// TwinCAT 3 PLC project DomeRunTime
// ProgramVersion: 3.1.4023.0
// libraries:
//   Tc2_Standard, * (Beckhoff Automation GmbH)
//   Tc2_System, * (Beckhoff Automation GmbH)
//   Tc2_Utilities, * (Beckhoff Automation GmbH)
//   Tc3_Module, * (Beckhoff Automation GmbH)
//   Tc2_SystemCX,3.3.6.0,Beckhoff Automation GmbH
// project tree:
//   GVLs/ GVL_Dome.TcGVL
//   / PlcTask.TcTTO
//   POUs/ FB_EventLog.TcPOU, MAIN.TcPOU, NewADSRoute.TcPOU
// real-time tasks:
//   TASK PlcTask: cycle T#10ms, priority 20, ADS port 350
// I/O:
//   DEVICE Gerät 2 (EtherCAT), AmsNetId 5.73.45.158.3.1
//     Klemme 1 (EK1200) [EK1200-5000 EtherCAT Netzteil (2A E-Bus)]
//       Klemme 2 (EL6021) [EL6021 Schnittstelle (RS422/485)]
//       Klemme 3 (EL2008) [EL2008 8K. Dig. Ausgang 24V, 0.5A]
//       Klemme 4 (EL1008) [EL1008 8K. Dig. Eingang 24V, 3ms]
//       Klemme 5 (EL9011) [EL9011 Endklemme]
// variable links:
//   DomeRunTime/DomeRunTime Instance <-> Device 2 (EtherCAT)/Term 1 (EK1200)/Term 3 (EL2008)
//     PlcTask Outputs/GVL_Dome.Flap_enable <-> Channel 1/Output
//     PlcTask Outputs/GVL_Dome.Flap_open <-> Channel 2/Output
//     PlcTask Outputs/GVL_Dome.Slit_enable <-> Channel 3/Output
//     PlcTask Outputs/GVL_Dome.slit_open <-> Channel 4/Output
//   DomeRunTime/DomeRunTime Instance <-> Device 2 (EtherCAT)/Term 1 (EK1200)/Term 4 (EL1008)
//     PlcTask Inputs/GVL_Dome.Input7 <-> Channel 7/Input

CONFIGURATION DomeRunTime
    RESOURCE PLC ON TwinCAT3
        TASK PlcTask(INTERVAL := T#10ms, PRIORITY := 20);
        PROGRAM MAIN WITH PlcTask : MAIN;
    END_RESOURCE
END_CONFIGURATION

// ---- GVLs/GVL_Dome.TcGVL
{attribute 'qualified_only'}
VAR_GLOBAL
	// enable flap hydraulics
	Flap_enable		AT%Q*:	BOOL;
	// open the flap, when true; close when false
	Flap_open		AT%Q*:	BOOL;
	// enable the slit motor
	Slit_enable		AT%Q*:	BOOL;
	// open the slit when true; close when false
	slit_open		AT%Q*:	BOOL;
	// Input signal 7 (0...7)
	Input7		AT%I*: BOOL;

	// ADS remote control word
	StatusWord		AT%MW0: WORD;
END_VAR

// ---- POUs/MAIN.TcPOU
PROGRAM MAIN
VAR
	// open flap command
	OpenFlap:	BOOL;
	// close flap command
	CloseFlap:	BOOL;
	// open slit command
	OpenSlit:	BOOL;
	// close slit command
	CloseSlit:	BOOL;
	// flap open state
	FlapOpen:	BOOL := TRUE; // assume Flap Open after restart
	// flap closed state
	FlapClosed:	BOOL := FALSE;
	// slit open state
	SlitOpen:	BOOL := TRUE; // assume Slit Open after restart
	// slit closed state
	SlitClosed:	BOOL := FALSE;
	// assume dome open, after power loss / reboot
	DomeOpen:	BOOL := FALSE;
	// dome closed state
	DomeClosed:	BOOL := FALSE;
	// control word is valid
	Valid:		BOOL;
	// timer to delay the flap
	FlapDelay: TON;
	// timer to delay the slit on reverse of direction
	SlitDelay:	TON;
	FlapTimer,
	SlitTimer:	TP := (PT := T#60S);
	FlapDone,
	SlitDone:	F_TRIG;
	SyncOut:	TON;
	TimeOut:	TON;
	WD_LED:		E_CX81x0_LED;
	ERR_LED:	E_CX81x0_LED;
	DomeOpenEvent:		FB_EventLog;
	DomeClosedEvent:	FB_EventLog;
	SyncEvent:		FB_Eventlog;
	TimeoutEvent:	FB_Eventlog;
	ADSErrorEvent:	FB_Eventlog;
	ReadCycle:	TON := (PT:=T#100MS);
	fbReadReq:	ADSREAD := ( NETID := '5.78.96.50.1.1', PORT := 851, TMOUT := DEFAULT_ADS_TIMEOUT );
	ControlWord: 	WORD;
	Busy:	BOOL;
	ADSError:	BOOL;
	ADSErrorID: UDINT;
END_VAR

(*
Dome Control Remote Unit CX8190
########################

The dome is controlled by the main PLC using the GVL_Dome.ControlWord,
which is used to exchange commands to open and close the slit and the flap
and to report wether the dome is open or closed.
*)
//NewADSRoute();
ReadCycle(IN := TRUE);
IF ReadCycle.Q THEN
	// read if the ADS command is busy
	fbReadReq(	READ := FALSE,
				BUSY => Busy,
				ERR =>	ADSError,
				ERRID => ADSErrorID);
	IF NOT Busy THEN
		fbReadReq(  IDXGRP := 16#4020, 
					IDXOFFS := 0, 
					LEN := SIZEOF(ControlWord), 
					DESTADDR := ADR(ControlWord),
					READ := TRUE,
					BUSY => Busy,
					ERR =>	ADSError,
					ERRID => ADSErrorID);
		ReadCycle(IN := FALSE);
	ELSE
		// reset the read command
		fbReadReq(READ := FALSE);
	END_IF
	IF NOT ADSError THEN // we have valid data
		Valid := 	ControlWord.0;
		OpenFlap := ControlWord.1;
		OpenSlit := ControlWord.2;
		CloseFlap := NOT ControlWord.1;
		CloseSlit := NOT ControlWord.2;
		ERR_LED := E_CX81x0_LED.eCX81x0_LED_RED_OFF;
	ELSE
		// reset the control word
		ControlWord := 0;
	END_IF
	
END_IF

// This is the sync timeout. If we loose the sync for 5 seconds, we issue a warning.
SyncOut(IN := NOT Valid, PT := T#5S);
IF SyncOut.Q THEN
	ERR_LED := E_CX81x0_LED.eCX81x0_LED_RED_FLASHING_200ms;
END_IF

// This is the watchdog timer. If we don't get a valid signal within n seconds, we issue to close the dome.
TimeOut(IN := NOT Valid, PT := T#30S);
IF TimeOut.Q THEN
	CloseFlap := NOT FlapClosed;
	CloseSlit := NOT SlitClosed;
	ERR_LED := E_CX81x0_LED.eCX81x0_LED_RED_ON;
END_IF

// cancel commands, if we know that the slot is closed
IF SlitClosed AND CloseSlit THEN
	CloseSlit := FALSE;
END_IF
IF SlitOpen AND OpenSlit THEN
	OpenSlit := FALSE;
END_IF
IF FlapClosed AND CloseFlap THEN
	CloseFlap := FALSE;
END_IF
IF FlapOpen AND OpenFlap THEN
	OpenFlap := FALSE;
END_IF

IF CloseSlit AND SlitTimer.Q THEN
	OpenSlit := FALSE;
	GVL_Dome.Slit_open := FALSE;
	WD_LED := E_CX81x0_LED.eCX81x0_LED_GREEN_FLASHING_500ms;
END_IF

IF OpenSlit AND SlitTimer.Q THEN
	GVL_Dome.Slit_open := TRUE;
	WD_LED := E_CX81x0_LED.eCX81x0_LED_RED_FLASHING_500ms;
END_IF

IF CloseFlap AND FlapTimer.Q  THEN
	OpenFlap := FALSE;
	GVL_Dome.Flap_open := FALSE;
	WD_LED := E_CX81x0_LED.eCX81x0_LED_GREEN_FLASHING_200ms;
END_IF

IF OpenFlap AND FlapTimer.Q THEN
	GVL_Dome.Flap_open := TRUE;
	WD_LED := E_CX81x0_LED.eCX81x0_LED_RED_FLASHING_200ms;
END_IF

// if we reverse the direction of the flap, wait n milliseconds, otherwise we blow the fuse
FlapDelay(  IN := OpenFlap OR CloseFlap,
			PT := T#1000MS);
// After an initial delay, enable the signal for n seconds to move the flap.
// we have to use different times for opening and closing especially at low temperatures
IF OpenFlap THEN
	FlapTimer.PT := T#30S;
ELSIF CloseFlap THEN
	FlapTimer.PT := T#60S;
END_IF			
FlapTimer(  IN := FlapDelay.Q,
			Q => GVL_Dome.Flap_enable);
// a falling edge of the enable signal indicates, that we are done
FlapDone(CLK := GVL_Dome.Flap_enable);
// deactivate open or close signal if enable becomes false;
IF FlapDone.Q THEN
	IF OpenFlap THEN
		FlapOpen 	:= TRUE;
		FlapClosed 	:= FALSE;
	ELSIF CloseFlap THEN
		FlapClosed 	:= TRUE;
		FlapOpen 	:= FALSE;
	END_IF
	OpenFlap := FALSE;
	CloseFlap := FALSE;
END_IF
			
// if we reverse the direction of the flap, wait n milliseconds, otherwise we blow the fuse
SlitDelay(  IN := OpenSlit OR CloseSlit, 
			PT := T#1000MS); 

// After an initial delay, enable the signal for n seconds to move the slit.			
SlitTimer(  IN := SlitDelay.Q,
			PT := T#70S,
			Q => GVL_Dome.Slit_enable); 
// a falling edge of the enable signal indicates, that we are done			
SlitDone(CLK := GVL_Dome.Slit_enable);

IF SlitDone.Q THEN
	IF OpenSlit THEN
		SlitOpen := TRUE;
		SlitClosed := FALSE;
	ELSIF CloseSlit THEN
		SlitClosed := TRUE;
		SlitOpen := FALSE;
	END_IF
	OpenSlit := FALSE;
	CloseSlit := FALSE;
END_IF

IF DomeOpen THEN
	WD_LED := E_CX81x0_LED.eCX81x0_LED_RED_ON;
END_IF
IF DomeClosed THEN
	WD_LED := E_CX81x0_LED.eCX81x0_LED_GREEN_ON;
END_IF

DomeOpen := FlapOpen AND SlitOpen;
DomeClosed := FlapClosed AND SlitClosed;

F_CX8190_LED_WD(eMode := WD_LED);
F_CX8190_LED_ERR(eMode := ERR_LED);

// set the status word
GVL_Dome.StatusWord.0 := TRUE;
GVL_Dome.StatusWord.1 := DomeOpen;
GVL_Dome.StatusWord.2 := DomeClosed;
GVL_Dome.StatusWord.3 := FlapOpen;
GVL_Dome.StatusWord.4 := FlapClosed;
GVL_Dome.StatusWord.5 := SlitOpen;
GVL_Dome.StatusWord.6 := SlitClosed;
GVL_Dome.StatusWord.7 := SyncOut.Q;
GVL_Dome.StatusWord.8 := TimeOut.Q;
GVL_Dome.StatusWord.9 := GVL_Dome.Input7;

DomeOpenEvent(
	Trigger := DomeOpen, 
	Level := ADSLOG_MSGTYPE_WARN,
	OnMessage := 'Dome is open.');

DomeClosedEvent(
	Trigger := DomeClosed, 
	Level := ADSLOG_MSGTYPE_HINT,
	OnMessage := 'Dome is closed.');

SyncEvent(
	Trigger := SyncOut.Q, 
	Level := ADSLOG_MSGTYPE_WARN,
	OnMessage := 'Synchronisation was lost.');
	
TimeoutEvent(
	Trigger := TimeOut.Q, 
	Level := ADSLOG_MSGTYPE_ERROR,
	OnMessage := 'Communication Timeout.',
	OffMessage := 'Communication reestablished');
	
ADSErrorEvent(
	Trigger := ADSError, 
	Level := ADSLOG_MSGTYPE_ERROR,
	FormatString := 'ADS Communication Error: %s',
	OnMessage := DWORD_TO_HEXSTR(ADSErrorID, 4, FALSE));

END_PROGRAM

// ---- POUs/FB_EventLog.TcPOU
FUNCTION_BLOCK FB_EventLog
VAR_INPUT
	Trigger:		BOOL;
	// ADSLOG_MSGTYPE_HINT or ADSLOG_MSGTYPE_WARN or ADSLOG_MSGTYPE_ERROR
	Level:			UDINT := ADSLOG_MSGTYPE_HINT;
	FormatString: 	STRING(255) := '%s';
	OnMessage: 		STRING(255) := '';
	OffMessage:		STRING(255) := '';
	OffLevel:		UDINT := ADSLOG_MSGTYPE_HINT;
END_VAR
VAR_OUTPUT
END_VAR
VAR
	LogonTrigger: R_TRIG;
	LogoffTrigger: F_TRIG;
END_VAR

LogonTrigger(CLK := Trigger);
LogoffTrigger(CLK := Trigger);
// in case the OffLevel is not set use the default Level Value
IF OffLevel = 0 THEN
	OffLevel := Level;
END_IF
IF LogonTrigger.Q AND LEN(OnMessage)>0 THEN
	ADSLOGSTR( Level OR ADSLOG_MSGTYPE_LOG, FormatString, OnMessage);
END_IF

IF LogoffTrigger.Q AND LEN(OffMessage)>0 THEN
	ADSLOGSTR( OffLevel OR ADSLOG_MSGTYPE_LOG, FormatString, OffMessage);
END_IF

END_FUNCTION_BLOCK

// ---- POUs/NewADSRoute.TcPOU
PROGRAM NewADSRoute
VAR
	// route 
	fbAddRoute  : FB_AddRouteEntry;
    // enable execution on first occurence
	bExecute    : BOOL := TRUE;
	// busy flag
    bBusy       : BOOL;
	// error flag
    bError      : BOOL;
	// error ID
    nErrID      : UDINT;
	// route parameters
    stRoute     : ST_AmsRouteEntry := ( sName := 'CX-4E6032',
                                        sNetID := '5.78.96.50.1.1',
                                        sAddress := '141.33.54.242',
                                        eTransport := eRouteTransport_TCP_IP );
END_VAR

fbAddRoute(	bExecute := bExecute,
			stRoute := stRoute,
			bBusy => bBusy,
			bError => bError,
			nErrID => nErrID);
// deactivate after first execution
bExecute := FALSE;

END_PROGRAM
